FUNCTION_BLOCK SludgeDischargeOC (* CAT Function Block Type *)
  (* Standard: 61499-2 *)
  (* Version 0.0, 6/7/2026, Schneider Electric, template *)
  PACKAGE SE.Nereda;
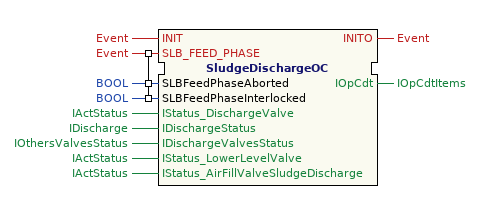
  EVENT_INPUT
    INIT;
    SLB_FEED_PHASE WITH SLBFeedPhaseAborted, SLBFeedPhaseInterlocked;
  END_EVENT
  EVENT_OUTPUT
    INITO;
  END_EVENT
  VAR_INPUT
    SLBFeedPhaseAborted : BOOL;
    SLBFeedPhaseInterlocked : BOOL;
  END_VAR
  SOCKETS
    IStatus_DischargeValve : IActStatus;
    IDischargeStatus : IDischarge;
    IDischargeValvesStatus : IOthersValvesStatus;
    IStatus_LowerLevelValve : IActStatus;
    IStatus_AirFillValveSludgeDischarge : IActStatus;
  END_SOCKETS
  PLUGS
    IOpCdt : IOpCdtItems;
  END_PLUGS
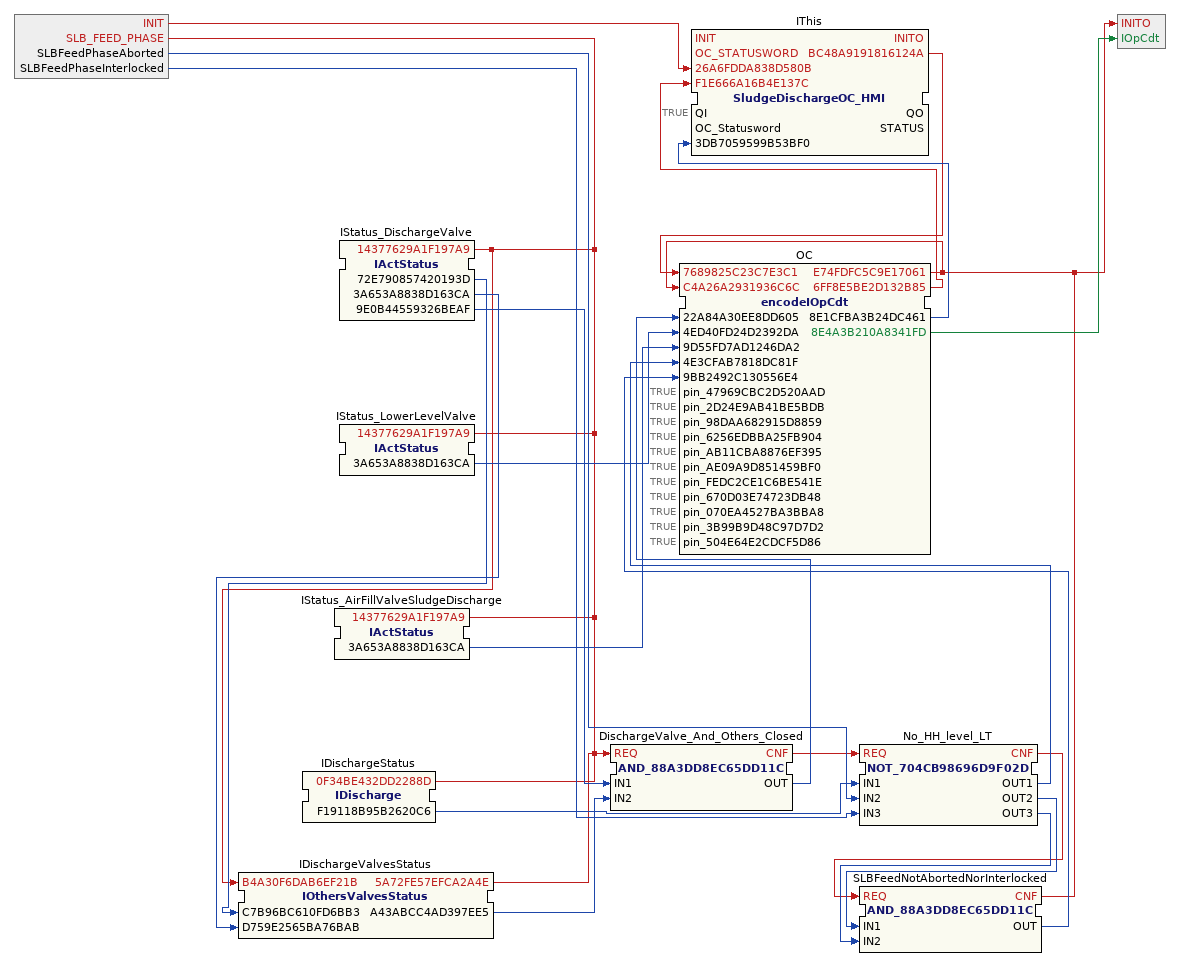
  (* 01 - FUNCTIONNAL INPUT INTERFACE *)
  (* 00 - INITIALIZATION *)
  (* 05 - LOGIC *)
  (* 06 - HMI INTERFACE *)
  (* 03 - FIELD INTERFACE *)
  (* 02 - FUNCTIONNAL OUTPUT INTERFACE *)
  (* Operating Condition Status *)
  (* Operating conditions : 1. Discharge valve AV41103 is available and valves for other reactors of the same line (AV4x103) is closed 2. Lower level valve AV41102 is closed. 3. Reserved, do not use 4. Phase ‘feed’ sludge buffer (1 for line A, 2 for line B) NOT aborted and NOT interlocked (1 for line A, 2 for line B) 5. Air fill valve sludge discharge AV41171 is closed *)
  (* Actuators Tags : - Feed valve :                                  AV4x101 - Lower level valve :                        AV4x102 - Air fill valve sludge discharge :    AV4x171 - Chemicals valve :                         AV4x108 - Discharge valve :                         AV4x103 - Vent aeration grid valve :             AV4x107 - Vent sludge grid valve :               AV4x172 *)
  FBS
    OC : encodeIOpCdt(pin_47969CBC2D520AAD := TRUE, pin_2D24E9AB41BE5BDB := TRUE, pin_98DAA682915D8859 := TRUE, pin_6256EDBBA25FB904 := TRUE, pin_AB11CBA8876EF395 := TRUE, pin_AE09A9D851459BF0 := TRUE, pin_FEDC2CE1C6BE541E := TRUE, pin_670D03E74723DB48 := TRUE, pin_070EA4527BA3BBA8 := TRUE, pin_3B99B9D48C97D7D2 := TRUE, pin_504E64E2CDCF5D86 := TRUE); (* You set the operating conditions. For the inputs that are not used set a constant to TRUE. *)
    IThis : SludgeDischargeOC_HMI(QI := TRUE);
    No_HH_level_LT : NOT_704CB98696D9F02D; {SET_ATTRIBUTE(Configuration.GenericFBType.InterfaceParams, Runtime.Standard#CNT:=3;OUT${CNT$}:BOOL,BOOL,BOOL)}
    DischargeValve_And_Others_Closed : AND_88A3DD8EC65DD11C; {SET_ATTRIBUTE(Configuration.GenericFBType.InterfaceParams, Runtime.Standard#CNT:=2;OUT:BOOL)}
    SLBFeedNotAbortedNorInterlocked : AND_88A3DD8EC65DD11C; {SET_ATTRIBUTE(Configuration.GenericFBType.InterfaceParams, Runtime.Standard#CNT:=2;OUT:BOOL)}
  END_FBS
  EVENT_CONNECTIONS
    INIT TO IThis.26A6FDDA838D580B;
    OC.E74FDFC5C9E17061 TO INITO;
    IStatus_DischargeValve.14377629A1F197A9 TO DischargeValve_And_Others_Closed.REQ;
    IStatus_DischargeValve.14377629A1F197A9 TO IDischargeValvesStatus.B4A30F6DAB6EF21B;
    IDischargeStatus.0F34BE432DD2288D TO DischargeValve_And_Others_Closed.REQ;
    IDischargeValvesStatus.5A72FE57EFCA2A4E TO DischargeValve_And_Others_Closed.REQ;
    OC.6FF8E5BE2D132B85 TO IThis.F1E666A16B4E137C;
    IThis.BC48A9191816124A TO OC.7689825C23C7E3C1;
    OC.E74FDFC5C9E17061 TO OC.C4A26A2931936C6C;
    IStatus_LowerLevelValve.14377629A1F197A9 TO DischargeValve_And_Others_Closed.REQ;
    IStatus_AirFillValveSludgeDischarge.14377629A1F197A9 TO DischargeValve_And_Others_Closed.REQ;
    SLB_FEED_PHASE TO DischargeValve_And_Others_Closed.REQ;
    DischargeValve_And_Others_Closed.CNF TO No_HH_level_LT.REQ;
    SLBFeedNotAbortedNorInterlocked.CNF TO OC.C4A26A2931936C6C;
    No_HH_level_LT.CNF TO SLBFeedNotAbortedNorInterlocked.REQ;
  END_CONNECTIONS
  DATA_CONNECTIONS
    IStatus_DischargeValve.72E790857420193D TO IDischargeValvesStatus.C7B96BC610FD6BB3;
    IStatus_DischargeValve.3A653A8838D163CA TO IDischargeValvesStatus.D759E2565BA76BAB;
    IStatus_DischargeValve.9E0B44559326BEAF TO DischargeValve_And_Others_Closed.IN1;
    IDischargeValvesStatus.A43ABCC4AD397EE5 TO DischargeValve_And_Others_Closed.IN2;
    OC.8E1CFBA3B24DC461 TO IThis.3DB7059599B53BF0;
    DischargeValve_And_Others_Closed.OUT TO OC.22A84A30EE8DD605;
    IStatus_LowerLevelValve.3A653A8838D163CA TO OC.4ED40FD24D2392DA;
    IStatus_AirFillValveSludgeDischarge.3A653A8838D163CA TO OC.9D55FD7AD1246DA2;
    IDischargeStatus.F19118B95B2620C6 TO No_HH_level_LT.IN1;
    No_HH_level_LT.OUT1 TO OC.4E3CFAB7818DC81F;
    SLBFeedPhaseAborted TO No_HH_level_LT.IN2;
    SLBFeedPhaseInterlocked TO No_HH_level_LT.IN3;
    No_HH_level_LT.OUT2 TO SLBFeedNotAbortedNorInterlocked.IN1;
    No_HH_level_LT.OUT3 TO SLBFeedNotAbortedNorInterlocked.IN2;
    SLBFeedNotAbortedNorInterlocked.OUT TO OC.9BB2492C130556E4;
  END_CONNECTIONS
  ADAPTER_CONNECTIONS
    OC.8E4A3B210A8341FD TO IOpCdt;
  END_CONNECTIONS
END_FUNCTION_BLOCK
